FUNCTION_BLOCK XTSHardware_V2 EXTENDS CyclicBase IMPLEMENTS I_Initialise
VAR
	XtsParts : ARRAY[1..SystemParameters.NumberOfParts] OF XtsPart;
	XtsTracks : ARRAY[1..SystemParameters.NumberOfTracks] OF XtsTrack;
	TrackOTCIDs: ARRAY [1..Tc3_XTS_Utility.TcIoXtsEnvironmentParameterList.MaxXtsTracksPerXpu] OF Tc3_XTS_Utility.OTCID;
	MyXPUInterface : Tc3_XTS_Utility.I_TcIoXtsProcessingUnit;
	MyXtsIoEnvVarRef : ITF_XTSIOEnvVarWrapper;
	XtsIoEnvInitialiseState : INT;
	i: INT;
END_VAR

METHOD Initialise : HRESULT
VAR_INPUT
END_VAR

VAR
	
END_VAR
CASE XtsIoEnvInitialiseState OF
	0:
		IF MyXtsIoEnvVarRef <> 0 THEN
			IF MyXtsIoEnvVarRef.IsInitialised() THEN
				XtsIoEnvInitialiseState := 1;
			END_IF
		END_IF
	1:
		IF MyXPUInterface.GetPartCount() = SystemParameters.NumberOfParts THEN
			FOR i := 1 TO SystemParameters.NumberOfParts DO
				XtsParts[i].MyXtsIoEnvInterface := MyXPUInterface.PartTcIo(UDINT_TO_UINT(i));
			END_FOR
			XtsIoEnvInitialiseState := 3;
		ELSE
			XtsIoEnvInitialiseState := 999;
		END_IF
	3:
		MyXPUInterface.GetTrackOids();
		TrackOTCIDs := MyXPUInterface.P_TrackOids;
		IF MyXPUInterface.GetTrackCount() = SystemParameters.NumberOfTracks THEN
			FOR i := 1 TO SystemParameters.NumberOfTracks DO
				XtsTracks[i].MyXtsIoEnvInterface := MyXPUInterface.TrackTcIo(UDINT_TO_UINT(i));
				XtsTracks[i].MyOTCID := TrackOTCIDs[i];
			END_FOR
			XtsIoEnvInitialiseState := 4;
		ELSE
			XtsIoEnvInitialiseState := 999;
		END_IF
	4:
		XtsIoEnvInitialiseState := 5;
		FOR i := 1 TO UDINT_TO_INT(MyXPUInterface.GetPartCount()) DO
			IF XtsParts[i].Initialise() <> 2 THEN
				XtsIoEnvInitialiseState := 4;
			END_IF
		END_FOR
	5:
		XtsIoEnvInitialiseState := 6;
		FOR i := 1 TO UDINT_TO_INT(MyXPUInterface.GetTrackCount()) DO
			IF XtsTracks[i].Initialise() <> 2 THEN
				XtsIoEnvInitialiseState := 5;
			END_IF
		END_FOR
	6:
		Initialise := 2;
END_CASE
END_METHOD

PROPERTY XtsIoEnvVarWrapper : itf_xtsioenvvarwrapper
GET
XtsIoEnvVarWrapper := MyXtsIoEnvVarRef;
END_GET
SET
MyXtsIoEnvVarRef := XtsIoEnvVarWrapper;
END_SET
END_PROPERTY

END_FUNCTION_BLOCK

(* stored: Version 1.1.0.1, ProductVersion 3.1.4024.12
   POU XTSHardware_V2: Id {2082c175-1a19-4a3f-b920-8dbd46477756}, SpecialFunc None
   Method Initialise: Id {95822be7-e433-46ff-bfc3-e4b3c51e2a74}
   Property XtsIoEnvVarWrapper: Id {9f0e6f27-b8f0-452c-b07d-d4d2a7ed1b3b}
   Get Get: Id {ef18a883-259a-46c5-ac1a-fd1d0138159b}
   Set Set: Id {3f18a9fd-c75b-45a9-b0a5-a4cb82b21b6b} *)
